# EPICS substitutions: iocBoot/ioc13bmc_laser/asynRecord.substitutions
file "$(ASYN)/db/asynRecord.db"
{
pattern
{P               R        PORT    ADDR    OMAX  IMAX}
{13BMC_Laser:   serial1   serial1    0     80     80}
{13BMC_Laser:   serial2   serial2    0     80     80}
}
